DATA_BLOCK "ST10_FB_S7connect_IDB"
{ S7_Optimized_Access := 'TRUE' }
VERSION : 0.1
NON_RETAIN
"ST10_FB_S7connect"

BEGIN

END_DATA_BLOCK

